PROGRAM MAIN
VAR
	fbSlicer : FB_Slicer;
	bStartButton : BOOL;
	bStopButton : BOOL;
	bContinueButton : BOOL;
	bHomeButton: BOOL;
	bEnginesOnButton : BOOL;
	bEnginesOffButton : BOOL;
	aStartingPosition : ARRAY[0..1] OF LREAL;
	aSlicingDimensions : ARRAY[0..1] OF LREAL;
	fVelocityOverride : LREAL := 80;
	fM1Position : LREAL;
	fM1sPosition : LREAL;
	fM2Position : LREAL;
	bEnginesLight : BOOL;
	bHomedLight : BOOL;
	bSlicingLight : BOOL;
	bStopLight : BOOL;
	bErrorLight : BOOL;
END_VAR

fbSlicer(bStartButton := bStartButton,
		 bStopButton := bStopButton,
		 bContinueButton := bContinueButton,
		 bHomeButton := bHomeButton,
		 bEnginesOnButton := bEnginesOnButton,
		 bEnginesOffButton := bEnginesOffButton,
		 aStartingPosition := aStartingPosition,
		 aSlicingDimensions := aSlicingDimensions,
		 fVelocityOverride := fVelocityOverride,
		 fM1Position => fM1Position,
		 fM1sPosition => fM1sPosition,
		 fM2Position => fM2Position,
		 bEnginesLight => bEnginesLight,
		 bHomedLight => bHomedLight,
		 bSlicingLight => bSlicingLight,
		 bStopLight => bStopLight,
		 bErrorLight => bErrorLight);

END_PROGRAM

(* stored: Version 1.1.0.1, ProductVersion 3.1.4024.12
   POU MAIN: Id {186648fb-a59e-43ef-bf6a-958903ba5b89}, SpecialFunc None *)
